{attribute addProperty BoxType "AX8206-0000-0041-0041"}
{attribute addProperty Id "Ch_B_ControlwordAT %Q*UINT162"}
{attribute addProperty CRC "1070582005"}
{attribute addProperty SizeInBites "16"}
{attribute addProperty SizeInBytes "2"}
TYPE Ch_B_AxisMain_Outputs_3FCFC8F5 :
STRUCT
	{attribute addProperty Name "Ch_B_Controlword"}
	Ch_B_Controlword AT %Q* : UINT;
END_STRUCT
END_TYPE

(* stored: Version 1.2.0.0, ProductVersion 3.1.4024.9
   DUT Ch_B_AxisMain_Outputs_3FCFC8F5: Id {90559942-8cac-40a2-a8cb-3b0acd288ae1} *)
